TYPE "GR_DQ_Config"
VERSION : 0.1
   STRUCT
      SOL_SD01_Signal : Bool;   // [O_G2_04.00] 2404CR01 - SOL_SD01_Signal
      SOL_SD02_Signal : Bool;   // [O_G2_04.01] 2404CR01 - SOL_SD02_Signal
      SOL_SD03_Signal : Bool;   // [O_G2_04.02] 2404CR01 - SOL_SD03_Signal
      SOL_SD04_Signal : Bool;   // [O_G2_04.03] 2404CR01 - SOL_SD04_Signal
      SOL_SD05_Signal : Bool;   // [O_G2_04.04] 2404CR02 - SOL_SD05_Signal
      "SEVOCONTROL ON" : Bool;   // [O_G2_04.05] 2404CR02 - SEVOCONTROL ON
      "PENDANT AUTO" : Bool;   // [O_G2_04.06]  - PENDANT AUTO
      "PENDANT TEACH" : Bool;   // [O_G2_04.07]  - PENDANT TEACH
      SPARE : Bool;   // [O_G2_04.08]  - SPARE
      SPARE_1 : Bool;   // [O_G2_04.09]  - SPARE
      SPARE_2 : Bool;   // [O_G2_04.10]  - SPARE
      SPARE_3 : Bool;   // [O_G2_04.11]  - SPARE
      SPARE_4 : Bool;   // [O_G2_04.12]  - SPARE
      SPARE_5 : Bool;   // [O_G2_04.13]  - SPARE
      SPARE_6 : Bool;   // [O_G2_04.14]  - SPARE
      SPARE_7 : Bool;   // [O_G2_04.15]  - SPARE
      TL_RED : Bool;   // [O_G2_05.00] 2154TL01 - TL_RED
      TL_YELLOW : Bool;   // [O_G2_05.01] 2154TL01 - TL_YELLOW
      TL_GREEN : Bool;   // [O_G2_05.02] 2154TL01 - TL_GREEN
      TL_BLUE : Bool;   // [O_G2_05.03] 2154TL01 - TL_BLUE
      BZ_CH1 : Bool;   // [O_G2_05.04] 2154BZ01 - BZ_CH1
      BZ_CH2 : Bool;   // [O_G2_05.05] 2154BZ01 - BZ_CH2
      BZ_CH3 : Bool;   // [O_G2_05.06] 2154BZ01 - BZ_CH3
      BZ_CH4 : Bool;   // [O_G2_05.07] 2154BZ01 - BZ_CH4
      SPARE_8 : Bool;   // [O_G2_05.08]  - SPARE
      SPARE_9 : Bool;   // [O_G2_05.09]  - SPARE
      SPARE_10 : Bool;   // [O_G2_05.10]  - SPARE
      SPARE_11 : Bool;   // [O_G2_05.11]  - SPARE
      SPARE_12 : Bool;   // [O_G2_05.12]  - SPARE
      SPARE_13 : Bool;   // [O_G2_05.13]  - SPARE
      SPARE_14 : Bool;   // [O_G2_05.14]  - SPARE
      SPARE_15 : Bool;   // [O_G2_05.15]  - SPARE
      Reserved_0 : Bool;
      Reserved_1 : Bool;
      Reserved_2 : Bool;
      Reserved_3 : Bool;
      Reserved_4 : Bool;
      Reserved_5 : Bool;
      Reserved_6 : Bool;
      Reserved_7 : Bool;
      Reserved_8 : Bool;
      Reserved_9 : Bool;
      Reserved_10 : Bool;
      Reserved_11 : Bool;
      Reserved_12 : Bool;
      Reserved_13 : Bool;
      Reserved_14 : Bool;
      Reserved_15 : Bool;
      Reserved_16 : Bool;
      Reserved_17 : Bool;
      Reserved_18 : Bool;
      Reserved_19 : Bool;
      Reserved_20 : Bool;
      Reserved_21 : Bool;
      Reserved_22 : Bool;
      Reserved_23 : Bool;
      Reserved_24 : Bool;
      Reserved_25 : Bool;
      Reserved_26 : Bool;
      Reserved_27 : Bool;
      Reserved_28 : Bool;
      Reserved_29 : Bool;
      Reserved_30 : Bool;
      Reserved_31 : Bool;
   END_STRUCT;

END_TYPE

